FUNCTION_BLOCK FB_MotionInterlocksGeneric IMPLEMENTS I_MotionInterlocksGeneric
VAR_INPUT
END_VAR
VAR_OUTPUT
END_VAR
VAR
    {attribute 'hide'}
    iMotionLogger 		: I_MotionLogger;
    {attribute 'hide'}
    iMotionInterlocksShareData : I_MotionInterlocksShareData;
    {attribute 'hide'}
    bAllForwardEnabled: BOOL:=FALSE;
    // Backward enable EPS summary
    {attribute 'hide'}
    bAllBackwardEnabled: BOOL:=FALSE;
    {attribute 'hide'}
    {attribute 'hide'}
    bPowerEnabled: BOOL:=FALSE;
   // If TRUE, we want to enable the motor independently of PMPS or other safety systems.
    bPowerSelf: BOOL:=FALSE;
    // TRUE if we have safety permission to move
    bSafetyReady: BOOL;
   // NC STO Input: TRUE if ok to move
    {attribute 'pytmc' := '
        pv: PLC:bHardwareEnable
        io: i
        field: ZNAM FALSE
        field: ONAM TRUE
        field: DESC TRUE if STO not hit
    '}
    bHardwareEnable AT %I*: BOOL ;

    // Used by the IOC to disable an axis
    {attribute 'pytmc' := '
        pv: PLC:bUserEnable
        io: io
        field: ZNAM DISABLE
        field: ONAM ENABLE
        field: DESC Used to disable power entirely for an axis
    '}
    bUserEnable: BOOL := TRUE;
    {attribute 'hide'}
    bEnable: BOOL;
    {attribute 'hide'}
    bExecute : BOOL;
    {attribute 'hide'}
    sMessage : STRING;
    {attribute 'hide'}
    bError : BOOL;
    {attribute 'hide'}
    nErrorID : UDINT;
    {attribute 'hide'}
    bMoveOk : BOOL;
    {attribute 'hide'}
    rtGlobalReset : R_TRIG;
    {attribute 'hide'}
    bInterlockEvent : BOOL;
END_VAR

IF ( iMotionInterlocksShareData = 0 ) OR ( iMotionLogger = 0) THEN
    // throw an exception
    RETURN;
END_IF

// read share
bPowerEnabled := iMotionInterlocksShareData.DriveEnable AND bHardwareEnable;
bPowerEnabled R= NOT bUserEnable;
// Moves are automatically allowed if no safety hooks. Otherwise, some other code will set this.
bSafetyReady S= bPowerSelf;

IF NOT bUserEnable THEN
    bError := TRUE;
    nErrorID:= 1;
    bMoveOk := FALSE;
    sMessage := 'User enable interlock triggered!';
ELSIF NOT bHardwareEnable THEN
    bError := TRUE;
    nErrorID:= 1;
    bMoveOk := FALSE;
    sMessage := 'Hardware enbale interlocks triggered!';
END_IF
// wait for global reset event to complete
rtGlobalReset(CLK:=iMotionInterlocksShareData.ResetDone);
IF rtGlobalReset.Q THEN
    bError := FALSE;
    nErrorID:= 0;
    sMessage:='';
END_IF

{warning 'add property implementation'}
PROPERTY Aborted : BOOL
GET
END_GET
END_PROPERTY

{warning 'add property implementation'}
PROPERTY Busy : BOOL
GET
END_GET
END_PROPERTY

{warning 'add property implementation'}
PROPERTY Done : BOOL
GET
END_GET
END_PROPERTY

{warning 'Add property implementation'}
PROPERTY Error : BOOL
GET
Error := bError;
END_GET
END_PROPERTY

{warning 'Add property implementation'}
PROPERTY ErrorID : UDINT
GET
ErrorID := nErrorID;
END_GET
END_PROPERTY

//FB_Init is always available implicitly and it is used primarily for initialization.
//The return value is not evaluated. For a specific influence, you can also declare the
//methods explicitly and provide additional code there with the standard initialization
//code. You can evaluate the return value.
METHOD FB_Init: BOOL
VAR_INPUT
    bInitRetains: BOOL; // TRUE: the retain variables are initialized (reset warm / reset cold)
    bInCopyCode: BOOL;  // TRUE: the instance will be copied to the copy code afterward (online change)

    iMotionLogger 		: I_MotionLogger;
    iMotionInterlocksShareData : I_MotionInterlocksShareData;
END_VAR
THIS^.iMotionLogger := iMotionLogger;
THIS^.iMotionInterlocksShareData := iMotionInterlocksShareData;
END_METHOD

{warning 'Add property implementation'}
PROPERTY InterlockEvent : BOOL
GET
InterlockEvent := bInterlockEvent;
END_GET
END_PROPERTY

{warning 'Add property implementation'}
PROPERTY Message : T_MAXSTRING
GET
END_GET
END_PROPERTY

{warning 'Add property implementation'}
PROPERTY MoveBackwardEnabled : BOOL
GET
END_GET
END_PROPERTY

{warning 'Add property implementation'}
PROPERTY MoveForwardEnabled : BOOL
GET
END_GET
END_PROPERTY

{warning 'Add property implementation'}
PROPERTY MoveOk : BOOL
GET
END_GET
END_PROPERTY

{warning 'Add property implementation'}
PROPERTY PowerEnabled : BOOL
GET
END_GET
END_PROPERTY

END_FUNCTION_BLOCK

(* stored: Version 1.1.0.1
   POU FB_MotionInterlocksGeneric: Id {b69073ed-2a55-41fc-84a9-b8fe79332e5e}, SpecialFunc None
   Property Aborted: Id {6c740eb9-40f2-43a5-962c-ed5e89b31929}
   Get Get: Id {48d77cf4-9dfd-41ed-aeba-f955cf151cfe}
   Property Busy: Id {d55880b8-fe7b-4ef7-86fb-317562726a5e}
   Get Get: Id {8f26a97a-35df-44f0-a763-d1f697bff7a3}
   Property Done: Id {19e5f483-e0b9-42ff-9068-b5fa5e63917b}
   Get Get: Id {a228592c-e271-409a-a873-134c01d2e742}
   Property Error: Id {21f5c9dd-d9f9-4fb7-a70a-688ad37ac74c}
   Get Get: Id {021721b1-8d55-49d6-a8cf-4547c5e3bcd2}
   Property ErrorID: Id {c58250f8-ae5a-4056-a2ed-503e8b03cb8d}
   Get Get: Id {a1817a62-dd31-4d18-8907-b880a900e971}
   Method FB_Init: Id {ee1048d7-3a0b-4701-a887-c2bc01c18e00}
   Property InterlockEvent: Id {8e1083ac-02c9-4b46-a759-679b00b2a867}
   Get Get: Id {9dcd64c3-1451-4b96-bcbf-7013a41cd9fd}
   Property Message: Id {fff95902-de95-4707-8ab7-164e983a966f}
   Get Get: Id {aa8e66bf-be37-477b-a097-6e499951d5ae}
   Property MoveBackwardEnabled: Id {73228441-2498-4cbf-b7a0-4009813e3963}
   Get Get: Id {f4731fcf-cdb2-4505-9bf3-b0970507bbd1}
   Property MoveForwardEnabled: Id {dbd2e5c0-7ee3-4d69-bfac-0c4778db19bb}
   Get Get: Id {b2fba177-14e5-4ae4-b487-6f6969050bec}
   Property MoveOk: Id {a6c854ac-10d2-4324-b515-25871c48273c}
   Get Get: Id {c6848f02-95c1-4045-9aa0-95260cab536e}
   Property PowerEnabled: Id {6a435248-a266-41ef-9b9c-8e0bf7663a4b}
   Get Get: Id {c27ac7b3-d93e-4dca-97d4-f9f71a18aff4} *)
